(* PLC project Unnamed, Unknown Unnamed 1 *)
(* stored: creationDateTime 2024-12-29T17:30:43, modificationDateTime 2024-12-29T18:49:43 *)

PROGRAM Bhaskara
  VAR
    A : REAL := 1.0;
    B : REAL := 0.0;
    C : REAL := -9.0;
    Xlinha : REAL;
    X2linha : REAL;
  END_VAR
  VAR  (* added by the conversion: wires and edge detectors of the diagram *)
    _SUB21_OUT : REAL;
    _SQRT6_OUT : REAL;
    _MUL17_OUT : REAL;
  END_VAR

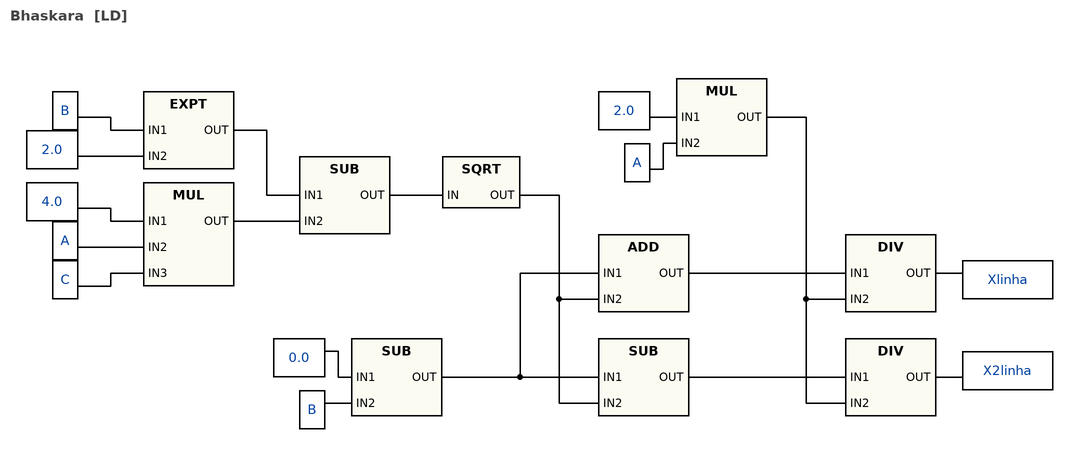
(* LD diagram, written out as Structured Text *)
_SUB21_OUT := 0.0 - B;
_SQRT6_OUT := SQRT(EXPT(B, 2.0) - 4.0 * A * C);
_MUL17_OUT := 2.0 * A;
Xlinha := (_SUB21_OUT + _SQRT6_OUT) / _MUL17_OUT;
X2linha := (_SUB21_OUT - _SQRT6_OUT) / _MUL17_OUT;
END_PROGRAM

CONFIGURATION Config0
  RESOURCE Res0 ON PLC
    TASK task0(INTERVAL := T#20ms, PRIORITY := 0);
    PROGRAM instance0 WITH task0 : Bhaskara;
  END_RESOURCE
END_CONFIGURATION
